{attribute 'GeneratedUsingTerminal: EK1100-0000-0018'}
{attribute addProperty BoxType "EK1100-0000-0018"}
{attribute addProperty Id "Beckhoff_ER7xxxEK1122Beckhoff_ER7xxxEK1122_0EBE6E72686"}
{attribute addProperty CRC "4291145287"}
{attribute addProperty Size "686"}
{attribute addProperty Name "Beckhoff ER7xxx"}
TYPE Beckhoff_ER7xxx_FFC5AE47 EXTENDS EK1100_1FC0878B :
STRUCT
	{attribute addProperty Name "Beckhoff ER7xxxEK1122"}
	{attribute addProperty PreviousPort "Beckhoff ER7xxx : B"}
	Beckhoff_ER7xxxEK1122 : Beckhoff_ER7xxxEK1122_0EBE6E72;
END_STRUCT
END_TYPE

(* stored: Version 1.2.0.0, ProductVersion 3.1.4024.11
   DUT Beckhoff_ER7xxx_FFC5AE47: Id {5dafd46d-334a-4790-b5c1-0273be6337e4} *)
